TYPE ST_AxisSafety :
STRUCT
	bTripped : BOOL;
	bSpeedLimited : BOOL;
	bLocalOnly : BOOL;
	iSafetyOutputGroup: INT;
	//Just ideas of axis specific info
END_STRUCT
END_TYPE

(* stored: Version 1.1.0.1, ProductVersion 3.1.4024.11
   DUT ST_AxisSafety: Id {eb178369-94a0-495a-8130-25faecb698cc} *)
